TYPE T_OUTER_Barcode : T_MaxString;
END_TYPE

(* stored: Version 1.1.0.1, ProductVersion 3.1.4024.15
   DUT T_OUTER_Barcode: Id {cfcea64c-fe4c-4188-ab59-9540fb8c4480} *)
